FUNCTION_BLOCK SPLIT_AL_INTO_AD (* this Function splits the 2 AD (DWORD) adapters from a AL (LWORD) *)
  (* Standard: 61499-2; Description: Copyright (c) 2026 Meisterschulen am Ostbahnhof SPDX-License-Identifier: EPL-2.0 *)
  (* Version 1.0, 2026-05-16, Franz Höpfinger, Meisterschulen am Ostbahnhof, initial API and implementation and/or initial documentation *)
  PACKAGE adapter::splitting;
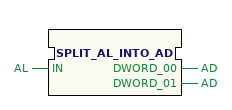
  SOCKETS
    IN : adapter::types::unidirectional::AL; (* LWORD Input *)
  END_SOCKETS
  PLUGS
    DWORD_00 : adapter::types::unidirectional::AD; (* DWord 0 *)
    DWORD_01 : adapter::types::unidirectional::AD; (* DWord 1 *)
  END_PLUGS
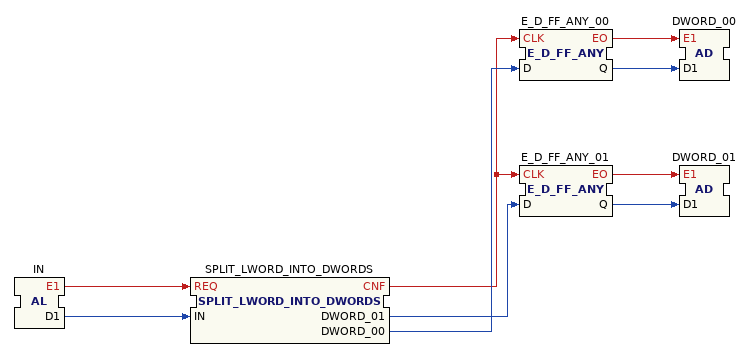
  FBS
    E_D_FF_ANY_00 : iec61499::events::E_D_FF_ANY;
    E_D_FF_ANY_01 : iec61499::events::E_D_FF_ANY;
    SPLIT_LWORD_INTO_DWORDS : eclipse4diac::utils::splitting::SPLIT_LWORD_INTO_DWORDS;
  END_FBS
  EVENT_CONNECTIONS
    IN.E1 TO SPLIT_LWORD_INTO_DWORDS.REQ;
    SPLIT_LWORD_INTO_DWORDS.CNF TO E_D_FF_ANY_00.CLK;
    SPLIT_LWORD_INTO_DWORDS.CNF TO E_D_FF_ANY_01.CLK;
    E_D_FF_ANY_00.EO TO DWORD_00.E1;
    E_D_FF_ANY_01.EO TO DWORD_01.E1;
  END_CONNECTIONS
  DATA_CONNECTIONS
    IN.D1 TO SPLIT_LWORD_INTO_DWORDS.IN;
    SPLIT_LWORD_INTO_DWORDS.DWORD_01 TO E_D_FF_ANY_01.D;
    SPLIT_LWORD_INTO_DWORDS.DWORD_00 TO E_D_FF_ANY_00.D;
    E_D_FF_ANY_00.Q TO DWORD_00.D1;
    E_D_FF_ANY_01.Q TO DWORD_01.D1;
  END_CONNECTIONS
END_FUNCTION_BLOCK
